INTERFACE I_StationInteraction

METHOD AddMover : BOOL
VAR_INPUT
	udiMoverID : UDINT;
END_VAR
END_METHOD

PROPERTY Cfg : reference to stStationCfg
GET
END_GET
END_PROPERTY

END_INTERFACE

(* stored: Version 1.1.0.1, ProductVersion 3.1.4024.11
   Itf I_StationInteraction: Id {187a8370-11e9-4c89-8477-36bd2151469a}
   Method AddMover: Id {a13cbc05-ee95-4977-aab6-3e712f1127f1}
   Property Cfg: Id {48b65226-185e-4e65-98d4-ea5c597e37f0}
   Get Get: Id {b8a03903-c3b2-41db-a830-e10b0d820684} *)
